Yaskawa INFORM job: CAL_MINI_RELATIVE.JBI

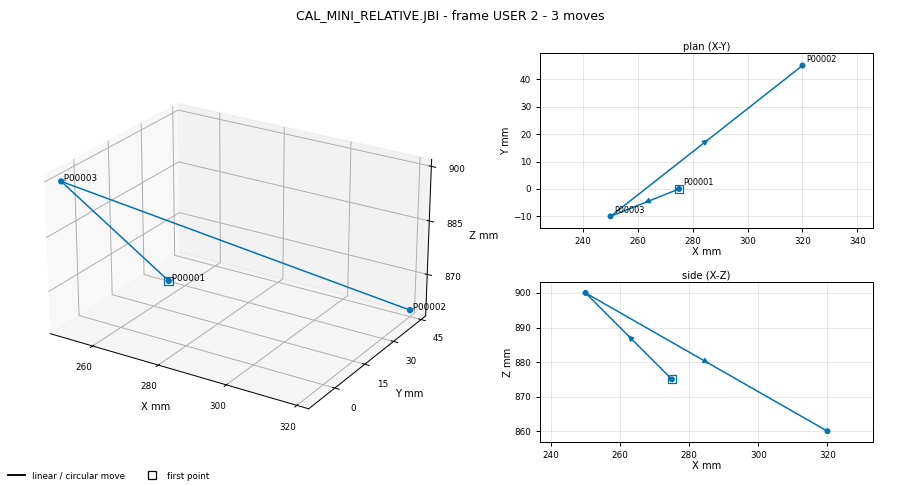
[picture p0: tool path of CAL_MINI_RELATIVE.JBI in frame USER 2, 3 of 3 moves have a stored position in this frame; points joined in program order, loops and branches not executed]
/JOB
//NAME CAL_MINI_RELATIVE
//POS
///NPOS 0,0,0,3,0,0
///TOOL 0
///POSTYPE USER
///USER 2
///RECTAN
///RCONF 1,0,0,0,0,0,0,0,0,0,0,0,0,0,0,0,0,0,0,0,0,0,0,0
P00001=275.000,0.000,875.000,180.0000,45.0000,0.0000
P00002=320.000,45.000,860.000,175.0000,40.0000,5.0000
P00003=250.000,-10.000,900.000,178.0000,42.0000,-2.0000
//INST
///DATE 2026/08/22 12:05
///ATTR SC,RW
///GROUP1 RB1
NOP
MSG "REL CAL — Phase B CART"
' Confirm cell clear, then CONTINUE
PAUSE
' CALSTEP:home
MSG "STEP_HOME"
' STEP_HOME
' PHASE B — CARTESIAN (relative / USER or BASE display)
' Home / safe pose (anchor)
PAUSE
MOVL P00001 V=50.0
' CALSTEP:uf2_rorg
MSG "STEP_UF2_RORG"
' STEP_UF2_RORG
' UF#2 S1 — RORG (origin)
PAUSE
MOVL P00003 V=50.0
' CALSTEP:joint_limit_S_plus
MSG "STEP_S_PLUS"
' STEP_S_PLUS
' S+ safe limit from home
PAUSE
MOVL P00002 V=50.0
MSG "REL CAL DONE — upload JBIs to PC"
END
